// Example 2 - ClothoidBallGap: ONE cam table, 18 points from FB_XtsBallCamBuilder.
//
//   Mover 1 = master, runs at constant velocity around the track.
//   Mover 2 = slave, follows Mover 1 through a cam table that covers one full lap (1500 mm).
//
// The two movers pinch one ball between them, like tongs: each mover carries a jaw BALL_OFFSET mm outboard of the
// track, and the table keeps the two jaws BALL_DISTANCE mm apart along the ball's path so the ball stays clamped
// through the curves. Mover 2 speeds up going into a curve and slows down coming out. The action BuildTable lets
// FB_XtsBallCamBuilder do the geometry.
//
// How to run (online view, with MAIN.eExample = ClothoidBallGap):  bStart -> watch eState -> bStop.   On Error: bReset.
// Watch fGapActual while it runs: 115 on the straights, dipping and rising through the curve transitions.
PROGRAM PRG_Example2
VAR CONSTANT
	// --- track geometry (mm) ---
	TRACK_LENGTH			: LREAL := 1500.0;	// = modulo factor of both mover axes
	CURVE_1_START			: LREAL := 250.0;
	CURVE_2_START			: LREAL := 1000.0;
	MODULE_LENGTH			: LREAL := 500.0;	// one 180 deg curve module (AT2050)

	// --- the ball clamped between the two movers ---
	BALL_DISTANCE			: LREAL := 115.0;	// mm between the two jaws, measured along the ball's path
	BALL_OFFSET				: LREAL := 103.03;	// mm the ball (and the jaws) sit outboard of the mover path
	TABLE_START				: LREAL := 180.0;	// master position of the first table point. Any point on straight 1
												// that keeps every ramp clear of the 1500 -> 0 wrap works (103 < x < 266).

	// --- demo dynamics ---
	MASTER_VELOCITY			: LREAL := 300.0;	// mm/s, Mover 1 while running
	POSITIONING_VELOCITY	: LREAL := 200.0;	// mm/s, Mover 2 while pre-positioning

	CAM_TABLE_ID			: MC_CAM_ID := 1;	// NC > Tables > Master 1 > Slave 1
	MAX_CAM_POINTS			: UDINT := 32;		// the builder writes 8 per curve + 2 = 18, the rest is room for tuning
	PLC_ERROR_ID			: UDINT := 16#FFFF_FFFF;	// not an NC error: the builder refused, see sTableError
END_VAR
VAR
	// --- commands: set TRUE in the online view, they reset themselves ---
	bStart				: BOOL;
	bStop				: BOOL;
	bReset				: BOOL;
	eState				: E_State;

	// --- cam table data: nCamPoints points, loaded into NC table CAM_TABLE_ID ---
	aCamPoints			: ARRAY[1..MAX_CAM_POINTS] OF MC_MotionFunctionPoint;
	nCamPoints			: UDINT;		// points actually used (18)
	stCamTable			: MC_CAM_REF;
	fbBuilder			: FB_XtsBallCamBuilder;	// computes the clothoid points

	// --- function blocks ---
	fbPowerMover1		: MC_Power;
	fbPowerMover2		: MC_Power;
	fbResetMover1		: MC_Reset;
	fbResetMover2		: MC_Reset;
	fbCamTableSelect	: MC_CamTableSelect;			// PLC array -> NC cam table
	fbReadTable			: MC_ReadCamTableSlaveDynamics;	// "where does the table want the slave for this master position?"
	fbMoveRelMover2		: MC_MoveRelative;
	fbCamIn				: MC_CamIn;
	fbMoveVeloMover1	: MC_MoveVelocity;
	fbHaltMover1		: MC_Halt;
	fbCamOut			: MC_CamOut;

	// --- live values worth watching ---
	fMover1Pos			: LREAL;	// modulo set position of Mover 1 (0..1500)
	fMover2Pos			: LREAL;	// modulo set position of Mover 2 (0..1500)
	fGapActual			: LREAL;	// how far Mover 2 is behind Mover 1 right now (along the track)
	fGapWanted			: LREAL;	// what the table asked for at coupling time
	fMasterInTable		: LREAL;	// fMover1Pos mapped into the master range of the table (TABLE_START .. +1500)
	bError				: BOOL;
	nErrorID			: UDINT;
	sTableError			: STRING(255);	// why the builder refused (nErrorID = PLC_ERROR_ID)
END_VAR

// update axis status every cycle
GVL_Axes.Mover1();
GVL_Axes.Mover2();

// live gap: Mover 1 position minus Mover 2 position, wrapped to 0..1500
fMover1Pos := GVL_Axes.Mover1.NcToPlc.ModuloSetPos;
fMover2Pos := GVL_Axes.Mover2.NcToPlc.ModuloSetPos;
fGapActual := fMover1Pos - fMover2Pos;
IF fGapActual < 0.0 THEN
	fGapActual := fGapActual + TRACK_LENGTH;
END_IF

CASE eState OF
	E_State.Idle:
		IF bStart THEN
			bStart := FALSE;
			eState := E_State.Enable;
		END_IF

	E_State.Enable:
		fbPowerMover1.Enable := TRUE;
		fbPowerMover1.Enable_Positive := TRUE;
		fbPowerMover1.Enable_Negative := TRUE;
		fbPowerMover2.Enable := TRUE;
		fbPowerMover2.Enable_Positive := TRUE;
		fbPowerMover2.Enable_Negative := TRUE;
		IF fbPowerMover1.Status AND fbPowerMover2.Status THEN
			eState := E_State.BuildTable;
		END_IF

	E_State.BuildTable:
		// fill the point array once, then hand it to the NC (overwrites cam table CAM_TABLE_ID)
		IF NOT fbCamTableSelect.Execute THEN
			BuildTable();
		END_IF
		IF nCamPoints > 0 THEN		// = 0: the builder refused, the error check below picks up sTableError
			fbCamTableSelect.Periodic := TRUE;		// one table = one lap, repeat forever
			fbCamTableSelect.CamTableID := CAM_TABLE_ID;
			fbCamTableSelect.Execute := TRUE;
			IF fbCamTableSelect.Done THEN
				fbCamTableSelect.Execute := FALSE;
				eState := E_State.ReadTable;
			END_IF
		END_IF

	E_State.ReadTable:
		// Mover 1 stays where it is. Ask the NC what slave position the table wants for it.
		// The table master runs from TABLE_START to TABLE_START + 1500, so a track position
		// below the table start is one lap further on in the table.
		IF NOT fbReadTable.Execute THEN
			fMasterInTable := fMover1Pos;
			IF fMasterInTable < TABLE_START THEN
				fMasterInTable := fMasterInTable + TRACK_LENGTH;
			END_IF
			fbReadTable.CamTableID := CAM_TABLE_ID;
			fbReadTable.MasterPosition := fMasterInTable;
		END_IF
		fbReadTable.Execute := TRUE;
		IF fbReadTable.Done THEN
			fbReadTable.Execute := FALSE;
			// table: slave = master - gap   ->   gap = master - slave
			fGapWanted := fMasterInTable - fbReadTable.SlavePosition;
			// Mover 1 stands still, so this relative move can never run into it:
			// positive = Mover 2 closes up from behind, negative = Mover 2 backs off a little
			fbMoveRelMover2.Distance := fGapActual - fGapWanted;
			eState := E_State.Preposition;
		END_IF

	E_State.Preposition:
		fbMoveRelMover2.Velocity := POSITIONING_VELOCITY;
		fbMoveRelMover2.Execute := TRUE;
		IF fbMoveRelMover2.Done THEN
			fbMoveRelMover2.Execute := FALSE;
			eState := E_State.CamIn;
		END_IF

	E_State.CamIn:
		fbCamIn.CamTableID := CAM_TABLE_ID;
		fbCamIn.StartMode := MC_STARTMODE_ABSOLUTE;		// table master axis = Mover 1 track position
		fbCamIn.MasterOffset := 0.0;
		fbCamIn.SlaveOffset := 0.0;
		fbCamIn.MasterScaling := 1.0;
		fbCamIn.SlaveScaling := 1.0;
		// let the NC pick the slave offset so Mover 2 never jumps at coupling.
		// After the pre-positioning above that offset is 0 (or whole laps), so the table gaps apply 1:1.
		fbCamIn.Options.SlaveScalingMode := MC_CAMSCALING_AUTOOFFSET;
		fbCamIn.Execute := TRUE;
		IF fbCamIn.InSync THEN
			fbCamIn.Execute := FALSE;
			eState := E_State.Run;
		END_IF

	E_State.Run:
		// only the master is commanded - the slave is driven by the cam
		fbMoveVeloMover1.Velocity := MASTER_VELOCITY;
		fbMoveVeloMover1.Direction := MC_Positive_Direction;
		fbMoveVeloMover1.Execute := TRUE;
		IF bStop THEN
			bStop := FALSE;
			fbMoveVeloMover1.Execute := FALSE;
			eState := E_State.Stopping;
		END_IF

	E_State.Stopping:
		fbHaltMover1.Execute := TRUE;
		IF fbHaltMover1.Done THEN
			fbHaltMover1.Execute := FALSE;
			eState := E_State.CamOut;
		END_IF

	E_State.CamOut:
		fbCamOut.Execute := TRUE;
		IF fbCamOut.Done THEN
			fbCamOut.Execute := FALSE;
			eState := E_State.Idle;
		END_IF

	E_State.Error:
		fbCamTableSelect.Execute := FALSE;
		fbReadTable.Execute := FALSE;
		fbMoveRelMover2.Execute := FALSE;
		fbCamIn.Execute := FALSE;
		fbMoveVeloMover1.Execute := FALSE;
		fbHaltMover1.Execute := FALSE;
		fbCamOut.Execute := FALSE;
		IF bReset THEN
			bReset := FALSE;
			fbResetMover1.Execute := TRUE;
			fbResetMover2.Execute := TRUE;
			eState := E_State.Resetting;
		END_IF

	E_State.Resetting:
		IF (fbResetMover1.Done OR fbResetMover1.Error) AND (fbResetMover2.Done OR fbResetMover2.Error) THEN
			fbResetMover1.Execute := FALSE;
			fbResetMover2.Execute := FALSE;
			bError := FALSE;
			nErrorID := 0;
			sTableError := '';
			eState := E_State.Idle;
		END_IF
END_CASE

// any error anywhere -> Error state
IF eState <> E_State.Error AND eState <> E_State.Resetting THEN
	IF GVL_Axes.Mover1.Status.Error THEN
		nErrorID := GVL_Axes.Mover1.Status.ErrorID;
	ELSIF GVL_Axes.Mover2.Status.Error THEN
		nErrorID := GVL_Axes.Mover2.Status.ErrorID;
	ELSIF fbPowerMover1.Error THEN
		nErrorID := fbPowerMover1.ErrorID;
	ELSIF fbPowerMover2.Error THEN
		nErrorID := fbPowerMover2.ErrorID;
	ELSIF sTableError <> '' THEN
		nErrorID := PLC_ERROR_ID;
	ELSIF fbCamTableSelect.Error THEN
		nErrorID := fbCamTableSelect.ErrorID;
	ELSIF fbReadTable.Error THEN
		nErrorID := fbReadTable.ErrorID;
	ELSIF fbMoveRelMover2.Error THEN
		nErrorID := fbMoveRelMover2.ErrorID;
	ELSIF fbCamIn.Error THEN
		nErrorID := fbCamIn.ErrorID;
	ELSIF fbMoveVeloMover1.Error THEN
		nErrorID := fbMoveVeloMover1.ErrorID;
	ELSIF fbHaltMover1.Error THEN
		nErrorID := fbHaltMover1.ErrorID;
	ELSIF fbCamOut.Error THEN
		nErrorID := fbCamOut.ErrorID;
	END_IF
	IF nErrorID <> 0 THEN
		bError := TRUE;
		eState := E_State.Error;
	END_IF
END_IF

// call every function block once per cycle
fbPowerMover1(Axis := GVL_Axes.Mover1);
fbPowerMover2(Axis := GVL_Axes.Mover2);
fbResetMover1(Axis := GVL_Axes.Mover1);
fbResetMover2(Axis := GVL_Axes.Mover2);
fbCamTableSelect(Master := GVL_Axes.Mover1, Slave := GVL_Axes.Mover2, CamTable := stCamTable);
fbReadTable();
fbMoveRelMover2(Axis := GVL_Axes.Mover2);
fbCamIn(Master := GVL_Axes.Mover1, Slave := GVL_Axes.Mover2);
fbMoveVeloMover1(Axis := GVL_Axes.Mover1);
fbHaltMover1(Axis := GVL_Axes.Mover1);
fbCamOut(Slave := GVL_Axes.Mover2);

ACTION BuildTable:
// One lap of Mover 1 (TABLE_START .. +1500) -> where Mover 2 has to be so that the two jaws stay
// BALL_DISTANCE apart along the ball's path and the ball stays clamped between them.
//
// FB_XtsBallCamBuilder does the geometry. The AT2050 curve module is not a plain half circle: its curvature
// ramps up over a short transition (a clothoid-like quintic), holds, and ramps down again. A jaw sitting
// BALL_OFFSET mm outboard of the track therefore travels further than the mover while the track is bending,
// so for the jaws to keep their distance the slave has to run faster than the master going into a curve
// and slower coming out. The builder writes 8 points per curve (ramp / plateau / ramp / line at the entry,
// mirrored at the exit) plus one point at each end of the table. See the FB header for the knot layout.
//
// Table master range 180..1680 instead of 0..1500: every ramp then lies inside the table and none of them
// straddles the 1500 -> 0 wrap of the track. The NC handles the lap mapping because the table is periodic.
sTableError := '';
nCamPoints := 0;

fbBuilder.fMasterStart		:= TABLE_START;
fbBuilder.fMasterEnd		:= TABLE_START + TRACK_LENGTH;
fbBuilder.fBallDistance		:= BALL_DISTANCE;
fbBuilder.fBallOffset		:= BALL_OFFSET;
fbBuilder.nCurves			:= 2;
fbBuilder.aCurveStart[1]	:= CURVE_1_START;
fbBuilder.aCurveStart[2]	:= CURVE_2_START;
fbBuilder.fModuleLength		:= MODULE_LENGTH;
// fTransLength, aEntryKnots, aExitKnots keep the FB defaults (tuned for 115 mm / 103 mm on AT2050 modules)
fbBuilder.pPoints			:= ADR(aCamPoints);
fbBuilder.nMaxPoints		:= MAX_CAM_POINTS;

IF NOT fbBuilder.Build() THEN
	sTableError := fbBuilder.sError;
	RETURN;
END_IF
nCamPoints := fbBuilder.nPoints;		// 18 (the builder terminates the last point itself)

// Slave goes from 65 (master 180) to 1565 (master 1680) = +1500 per lap, the same "cyclic cam with lift"
// as the ConstantGap table of example 1, so Mover 2 keeps going around with Mover 1.

// describe the array to the NC
stCamTable.pArray		:= ADR(aCamPoints);
stCamTable.ArraySize	:= nCamPoints * SIZEOF(MC_MotionFunctionPoint);
stCamTable.TableType	:= MC_TABLETYPE_MOTIONFUNCTION;
stCamTable.NoOfRows		:= nCamPoints;
stCamTable.NoOfColumns	:= 1;
END_ACTION

END_PROGRAM

(* stored: Version 1.1.0.1
   POU PRG_Example2: Id {4f8d1ff5-9d58-4f77-9655-f1c94407d59e}, SpecialFunc None
   Action BuildTable: Id {be6e4ebf-3b96-495f-a557-9538384560a4} *)
